FUNCTION_BLOCK FB_TestSplit EXTENDS TcUnit.FB_TestSuite

testSplit();

METHOD testSplit : BOOL
VAR
	sToSplit		: STRING(255) := 'Hello,this,is,split,test';
	sSplit			: ARRAY[0..Parameters.iSplitArraySize] OF STRING(255);
	sExpected		: ARRAY[0..Parameters.iSplitArraySize] OF STRING(255) := ['Hello', 'this', 'is', 'split', 'test'] ;
	
	i				: INT;
END_VAR
Test('testSplit');
// Arrange

// Act
sSplit := F_STRING_SPLIT(sToSplit, ',');

// Assert
FOR i := 0 TO Parameters.iSplitArraySize DO
	AssertEquals_STRING( Expected := sExpected[i],
				  Actual := sSplit[i],
				  Message := CONCAT('testSplit Failed to split : ', sToSplit));
END_FOR
			 
			 
TEST_FINISHED();
END_METHOD

END_FUNCTION_BLOCK

(* stored: Version 1.1.0.1, ProductVersion 3.1.4024.9
   POU FB_TestSplit: Id {c399aa91-0228-4585-b4f7-87e722765771}, SpecialFunc None
   Method testSplit: Id {71d86309-488d-4c73-9afa-751071041933} *)
